(* PLC project Tc2_Utilities.F_EuropeanLocalTime Demo, tc3-libraries-kb TwinCAT 3.1 *)
(* stored: creationDateTime 2026-05-10T12:00:00, modificationDateTime 2026-05-10T12:00:00 *)

PROGRAM P_Demo_F_EuropeanLocalTime
  VAR
    rResult : TIMESTRUCT;  (* F_EuropeanLocalTime 的返回值 *)
    bRun : BOOL;  (* 触发一次调用 *)
    stUtc : TIMESTRUCT;  (* 测试用本地变量 *)
    bDST : BOOL;  (* 测试用本地变量 *)
    out_bDaylightSavingTime : BOOL;  (* VAR_OUTPUT bDaylightSavingTime *)
  END_VAR

            // ============================================================
// Tc2_Utilities.F_EuropeanLocalTime 演示程序（FUNCTION）
// ============================================================
// 验证步骤：
//   1. 引用 Tc2_Utilities（及类型所在依赖库 Tc2_System / Tc2_Standard）
//   2. 编译 + 登录
//   3. 强制 bRun := TRUE 一个周期
//   4. 观察 rResult 应为 本地时（DST 期 +120 分钟）
// ============================================================

stUtc.wYear := 2024; stUtc.wMonth := 7; stUtc.wDay := 15; stUtc.wHour := 10;
IF bRun THEN
    rResult := F_EuropeanLocalTime(stUtc, 60);
    bRun := FALSE;
END_IF;

          
END_PROGRAM
